// TIA Portal V21 export
TYPE "Std_PrmAllarmeStd"
   STRUCT
      Abilitato : Bool;   // 1 = Allarme presente / 0 = Allarme non presente
      Stato : Bool;   // 1 = Allarme Attivo / 0 = Allarme non attivo
      Silenziato : Bool;   // 1 = Allarme silenziato / 0 = Allarme non silenziato
      EnWarnHmi : Bool;   // Abilitazione dell'allarme ad essere mostrato nella lista HMI
      EnCadutaCiclo : Bool;   // Abilitazione dell'allarme a far cadere il ciclo automatico
   END_STRUCT;
END_TYPE
